{attribute 'pack_mode' := '2'}
TYPE ST_MOVER_STATE :
STRUCT
  State           : E_MOVER_STATE;  // ST_MOVER_CTRL.Cmd with added E_PROGRESS
  MasterId        : USINT;            // mirror NC AxisId of Master axis
END_STRUCT
END_TYPE

(* stored: Version 1.1.0.1, ProductVersion 3.1.4026.13
   DUT ST_MOVER_STATE: Id {2ceabe02-3e09-480c-afb7-f28bb73cc94a} *)
